// TIA Portal V15.1 export
// export: Created 2019-08-14T06:26:55.3891978Z, ExportSetting None, DisplayName Totally Integrated Automation Portal, DisplayVersion V15.1, DisplayName TIA Portal Openness, DisplayVersion V15.1, DisplayName STEP 7 Professional, DisplayVersion V15.1, DisplayName STEP 7 Safety, DisplayVersion V15.1, DisplayName WinCC Advanced, DisplayVersion V15.1
FUNCTION_BLOCK "Skill_#SKILL_NAME#"   // FB13, SCL
{ S7_Optimized_Access := 'TRUE' }
// stored: MemoryReserve 100, SetENOAutomatically False
   VAR_INPUT
      ModulToSkill : "typeModulSkillInterface_IN";
   END_VAR
   VAR_OUTPUT
      SkillToModul : "typeModulSkillInterface_OUT";
   END_VAR
   VAR
      State { S7_SetPoint := 'True'} : UInt;
      StateOfExecute : UInt;
      ResultTrigger : DInt;   // value increases at new result available
      ResultFeched : Bool;   // true= result fechted
      oldResultTrigger : DInt;
      NextStep : Bool;
      Parameter_In : "type#SKILL_NAME#StartParameter_In";
      Parameter_Out : "type#SKILL_NAME#GetResultParameter_Out";
      statErrorId { S7_SetPoint := 'True'} : Int;
      ResultAcknowledge : Bool;
      StartByMES { S7_SetPoint := 'True'} : Bool;
      rtStart : R_TRIG;
      rtStop : R_TRIG;
      rtAbort : R_TRIG;
      rtReset : R_TRIG;
      rtStep : R_TRIG;
      rtNextStep : R_TRIG;
      Start : "#SKILL_NAME#_Start";
      GetResult : "#SKILL_NAME#_GetResult";
   END_VAR
   VAR CONSTANT
      StateInit : UInt := 0;
      StateIdle : UInt := 100;
      StateExecute : UInt := 200;
      StateCompleting : UInt := 300;
      StateComplete : UInt := 400;
      StateProvideResult : UInt := 8998;
      StatePreDone : UInt := 8999;
      StateDone : UInt := 9000;
      StateError : UInt := 9001;
      ExecuteSkill : UInt := 100;
      ERRORID_NO_ERROR : Int := 0;
   END_VAR
BEGIN
   (*******************************************************************
   // Description
   //   #####
   // Version
   // V0.01 2019-07-24 

   // Authors
   // Michael Elting evtl. durch SiOME Version ersetzen
   //
   // © Alle Rechte vorbehalten/All rights reserved, Siemens AG, 2019
   *******************************************************************)

   REGION ##Enabled
       IF NOT #ModulToSkill.Enable THEN
           RETURN;
       END_IF;
   END_REGION

   REGION ##Init or Reset
       IF #ModulToSkill.Init OR #ModulToSkill.Reset THEN
           #State := 0;
           #ResultTrigger := 0;
           #statErrorId := #ERRORID_NO_ERROR;

           #SkillToModul.TaskBusy := FALSE;
           #SkillToModul.TaskDone := FALSE;
           #SkillToModul.TaskError := FALSE;
           #SkillToModul.TaskReady := FALSE;
           #SkillToModul.TaskInitPos := FALSE;
       END_IF;
   END_REGION

   REGION OPC_UA_Method_Calls
       REGION Start Skill
           #Start(ModulToSkill:=#ModulToSkill,
                  SkillToModul:=#SkillToModul,
                  StartSkill := #StartByMES,
                  Parameter := #Parameter_In);
       END_REGION

       REGION Provide Results
           #GetResult(Automatic := #ModulToSkill.Automatic,
                      ResultTrigger := #ResultTrigger,
                      ResultFeched:=#ResultFeched,
                      Parameter_Out := #Parameter_Out);
       END_REGION
   END_REGION

   REGION ##Edge detection
       #rtStart(CLK := #StartByMES OR #ModulToSkill.Start);
       #rtStop(CLK := #ModulToSkill.Stop);
       #rtReset(CLK := #ModulToSkill.Reset);
       #rtNextStep(CLK := #ModulToSkill.Step);
   END_REGION

   REGION ##NextState
       #NextStep := (#ModulToSkill.Automatic) OR
       (#ModulToSkill.SingleStep AND #rtNextStep.Q);
   END_REGION

   REGION StateMachine
       CASE #State OF
           #StateInit: // Init skill state maschine
               REGION Init
               (*
               Enter here code for init skill purpose
               *)
                   #State := + #StateIdle;
               END_REGION


           #StateIdle: // wait for incomming skill request
               REGION IDLE

                   IF #rtStart.Q THEN
                       #statErrorId := 0;
                       #SkillToModul.TaskBusy := TRUE;
                       #SkillToModul.TaskDone := FALSE;
                       #SkillToModul.TaskError := FALSE;
                       #State := #StateExecute;
                   END_IF;
               END_REGION

           #StateExecute:
               #State += 1;
               // CASE #StateOfExecute OF
               //     #ExecuteSkill:  // Statement section case 1
               //         // do Execution
               //         // 

               //         IF true THEN
               //             ;
               //         END_IF;
               //         ;
               //     #NextStep:  // Statement section case 2 to 4
               //         ;
               //     ELSE  // Statement section ELSE
               //         ;
               // END_CASE;
               ;

           201..8997:  // States to do skill actions
               #State += 1;

           #StateProvideResult:
               REGION Provide Result
                   // Trigger Get Values
                   #ResultTrigger += 1;
                   #ResultFeched := FALSE;
                   #Parameter_Out.ErrorId := #ERRORID_NO_ERROR;
                   #State := #StatePreDone;
                   ;
               END_REGION

           #StatePreDone:
               REGION ##PreDone
                   IF #ResultFeched THEN
                       #State := #StateDone;
                   END_IF;
               END_REGION


           #StateDone:
               REGION ##Done
                   #SkillToModul.TaskBusy := FALSE;
                   #SkillToModul.TaskDone := TRUE;
                   IF #statErrorId <> #ERRORID_NO_ERROR THEN
                       #SkillToModul.TaskError := TRUE;
                       #Parameter_Out.ErrorId := #statErrorId;
                       #State := #StateError;
                   ELSE
                       #State := #StateIdle;
                   END_IF;
               END_REGION


           #StateError:
               REGION ##Error
                   #SkillToModul.TaskBusy := FALSE;
                   #SkillToModul.TaskDone := TRUE;
                   #SkillToModul.TaskError := TRUE;
                   ; //wait FOR #Reset OR Init
               END_REGION

           ELSE  // Statement section ELSE
               #State := #StateError;
       END_CASE;

   END_REGION

   REGION ##State Mapping

   END_REGION
END_FUNCTION_BLOCK
